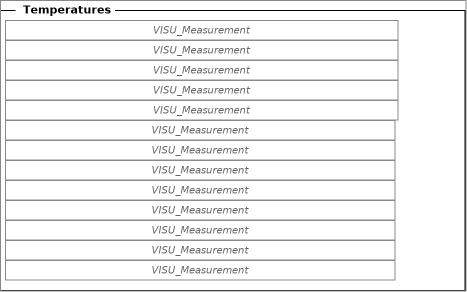
VISUALIZATION VISU_TelemetryTemperatures  // 467x292
VAR_IN_OUT
    ref : TelemetryTemperatures;
	widget : TelemetryTemperaturesWidget;
END_VAR
    Label (20,0 90x20), "Temperatures"
    Line (465,290) (465,10)
        p2175578022: widget.actualStatus.color.bg
    Frame (5,20 393x20)
        shows VISU_Measurement(widget := widget.m1)
    Frame (5,40 393x20)
        shows VISU_Measurement(widget := widget.mirrorCell)
    Frame (5,60 393x20)
        shows VISU_Measurement(widget := widget.m2)
    Frame (5,80 393x20)
        shows VISU_Measurement(widget := widget.m2Electronics)
    Frame (5,100 393x20)
        shows VISU_Measurement(widget := widget.topTube)
    Frame (5,120 390x20)
        shows VISU_Measurement(widget := widget.centreTube)
    Frame (5,140 390x20)
        shows VISU_Measurement(widget := widget.fork)
    Frame (5,160 390x20)
        shows VISU_Measurement(widget := widget.nasmythAir)
    Frame (5,180 390x20)
        shows VISU_Measurement(widget := widget.rem)
    Frame (5,200 390x20)
        shows VISU_Measurement(widget := widget.rpm)
    Frame (5,220 390x20)
        shows VISU_Measurement(widget := widget.hermesTelescopeAdapter)
    Frame (5,240 390x20)
        shows VISU_Measurement(widget := widget.topAir)
    Frame (5,260 390x20)
        shows VISU_Measurement(widget := widget.insideTube)
    Line (115,10) (465,10)
        p2175578022: widget.actualStatus.color.bg
    Line (0,10) (15,10)
        p2175578022: widget.actualStatus.color.bg
    Line (0,290) (0,10)
        p2175578022: widget.actualStatus.color.bg
    Line (0,290) (465,290)
        p2175578022: widget.actualStatus.color.bg
END_VISUALIZATION

(* stored: Version 1.1.0.1, ProductVersion 3.1.4019.2
   Visu VISU_TelemetryTemperatures: Id {8c30eea0-9487-4515-b4a9-904dca7071c0} *)
